FUNCTION_BLOCK Emitr
  (* Standard: 61499-2 *)
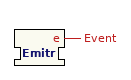
  EVENT_OUTPUT
    e;
  END_EVENT
END_FUNCTION_BLOCK
(* other elements stored in the file *)
(* Autogenerate Language=C RunText=me->outputEvents.event.e = 1; *)
